INTERFACE ITcoInspectionGroupInspect EXTENDS IInspector

METHOD Inspect : ITcoInspectionGroupInspect
VAR_INPUT
    Inspector : IInspector;
END_VAR
END_METHOD

END_INTERFACE

(* stored: Version 1.1.0.1, ProductVersion 3.1.4024.9
   Itf ITcoInspectionGroupInspect: Id {0107fc9a-abbf-041f-04a8-2d57c254b027}
   Method Inspect: Id {4c025f4a-bace-0217-36db-8dbb6ef5791f} *)
